SUBAPPLICATION OPC_TO_AR2 (* Nur OPC-UA (kein VT-Eingabefeld): Remote-Wert lesen (Subscribe) und als AR2 (bidirektional) an einen Consumer weiterreichen. Was der Consumer zurueckechot (z.B. CALIBRATE.ZERO/.SPAN Boot-/Live-Wert) wird per Publish auf dieselbe Remote-Adresse zurueckgemeldet. *)
  (* Standard: 61499-2; Description: Copyright (c) 2026 Meisterschulen am Ostbahnhof This program and the accompanying materials are made available under the terms of the Eclipse Public License 2.0 which is available at https://www.eclipse.org/legal/epl-2.0/ SPDX-License-Identifier: EPL-2.0 *)
  (* Version 1.0, 2026-08-31, Franz Höpfinger, Meisterschulen am Ostbahnhof, OPC-UA-only sibling of NumericValue_TO_AR2 - no VT object involved, purely remote read+echo via AR2 *)
  PACKAGE MyLib::sys;
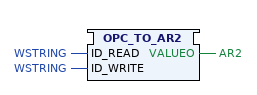
  VAR_INPUT
    ID_READ : WSTRING; (* Remote-Subscribe-Adresse (REAL, ACTION=SUBSCRIBE) *)
    ID_WRITE : WSTRING; (* Remote-Echo-Adresse (REAL, ACTION=PUBLISH) - meldet zurueck, was der Consumer gerade als aktuellen/persistierten Wert liefert *)
  END_VAR
  PLUGS
    VALUEO : adapter::types::bidirectional::AR2;
  END_PLUGS
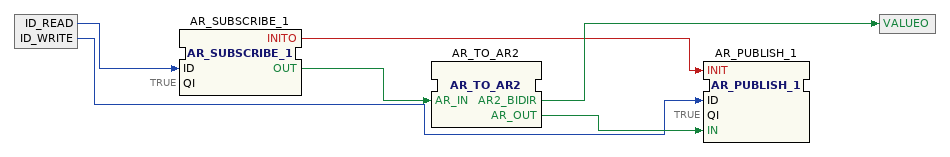
  FBS
    AR_SUBSCRIBE_1 : adapter::net::AR_SUBSCRIBE_1(QI := TRUE);
    AR_TO_AR2 : adapter::conversion::bidirectional::AR_TO_AR2;
    AR_PUBLISH_1 : adapter::net::AR_PUBLISH_1(QI := TRUE);
  END_FBS
  EVENT_CONNECTIONS
    AR_SUBSCRIBE_1.INITO TO AR_PUBLISH_1.INIT;
  END_CONNECTIONS
  DATA_CONNECTIONS
    ID_READ TO AR_SUBSCRIBE_1.ID;
    ID_WRITE TO AR_PUBLISH_1.ID;
  END_CONNECTIONS
  ADAPTER_CONNECTIONS
    AR_SUBSCRIBE_1.OUT TO AR_TO_AR2.AR_IN;
    AR_TO_AR2.AR2_BIDIR TO VALUEO;
    AR_TO_AR2.AR_OUT TO AR_PUBLISH_1.IN;
  END_CONNECTIONS
END_SUBAPPLICATION
